{attribute addProperty BoxType "EL5021-0000-0019"}
{attribute addProperty Id "StatusAT %I*Status_16FD7F051621Counter_valueAT %I*UDINT32417Latch_valueAT %I*UDINT32418"}
{attribute addProperty CRC "3123730512"}
{attribute addProperty SizeInBites "80"}
{attribute addProperty SizeInBytes "10"}
TYPE ENC_Status_BA305850 :
STRUCT
	{attribute addProperty Name "Status"}
	Status AT %I* : Status_16FD7F05;
	{attribute addProperty Name "Counter_value"}
	Counter_value AT %I* : UDINT;
	{attribute addProperty Name "Latch_value"}
	Latch_value AT %I* : UDINT;
END_STRUCT
END_TYPE

(* stored: Version 1.2.0.0, ProductVersion 3.1.4024.9
   DUT ENC_Status_BA305850: Id {121c8434-c928-4719-b11b-5d9f6ceeeb9b} *)
